// TIA Portal V19 export
ORGANIZATION_BLOCK "Startup"   // OB2203, LAD, Startup
TITLE = "Complete Restart"
// stored: AutoNumber false, Namespace Unit2.EM1, SetENOAutomatically false
   VAR_INPUT
      LostRetentive : Bool;   // True if retentive data are lost
      LostRTC : Bool;   // True if date and time are lost
   END_VAR
BEGIN

REGION Network 2 (SCL)
   IF LEN(IN := "Unit2.EM1.Config".em.referenceDesignator.parent) <> 0 THEN
       "Unit2.EM1.Config".em.referenceDesignator.combined := CONCAT_WSTRING(IN1 := "Unit2.EM1.Config".em.referenceDesignator.parent, IN2 := WSTRING#'.', IN3 := "Unit2.EM1.Config".em.referenceDesignator.relative);
   ELSE
       "Unit2.EM1.Config".em.referenceDesignator.combined := "Unit2.EM1.Config".em.referenceDesignator.relative;
   END_IF;
END_REGION
END_ORGANIZATION_BLOCK
